PROGRAM Halt_Axis
VAR
	fbHalt: MC_Halt;
	HaltPB: BOOL;
	HaltDone: BOOL;
END_VAR

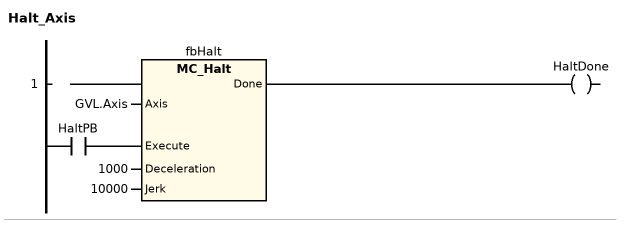
// NETWORK 1
fbHalt(Axis := GVL.Axis, Execute := HaltPB, Deceleration := 1000, Jerk := 10000); // MC_Halt
HaltDone := fbHalt.Done;

END_PROGRAM

(* stored: Version 1.1.0.1, ProductVersion 3.1.4024.12
   POU Halt_Axis: Id {35714abc-9861-4a45-9a29-c7aa268d480f}, SpecialFunc None *)
